{attribute 'qualified_only'}
{attribute 'strict'}
{attribute 'to_string'}
TYPE E_Result :
(
	invalid := 0,
	inProgress,
	done,
	aborted
);
END_TYPE

(* stored: Version 1.1.0.1
   DUT E_Result: Id {d16560f9-d408-452f-8c8d-282023243f25} *)
